FUNCTION_BLOCK ABSTRACT FB_Cyclic EXTENDS FB_Base IMPLEMENTS I_Cyclic
VAR
	_InitCompleted : BOOL;
END_VAR

{warning 'add method implementation '}
METHOD CyclicLogic : BOOL
END_METHOD

{warning 'add property implementation'}
PROPERTY InitCompleted : BOOL
GET
InitCompleted := _InitCompleted;
END_GET
END_PROPERTY

END_FUNCTION_BLOCK

(* stored: Version 1.1.0.1, ProductVersion 3.1.4024.14
   POU FB_Cyclic: Id {b52f827f-edb9-4b5a-b1d9-3112b134d109}, SpecialFunc None
   Folder Methods: Id {091563a2-2114-4d7e-9a99-1aa5cdaa3f65}
   Folder Properties: Id {e6fe3d3a-8188-4c70-bd35-6a995c218a13}
   Method CyclicLogic: Id {25d97232-7a76-4aec-bdd5-31f940f4d8f8}
   Property InitCompleted: Id {e3b13183-b852-4644-aecd-ea5e517dc9f4}
   Get Get: Id {81bd1a58-ed2a-43f6-9626-1039008d36a6} *)
